PROGRAM T01_CONTROL
VAR
END_VAR

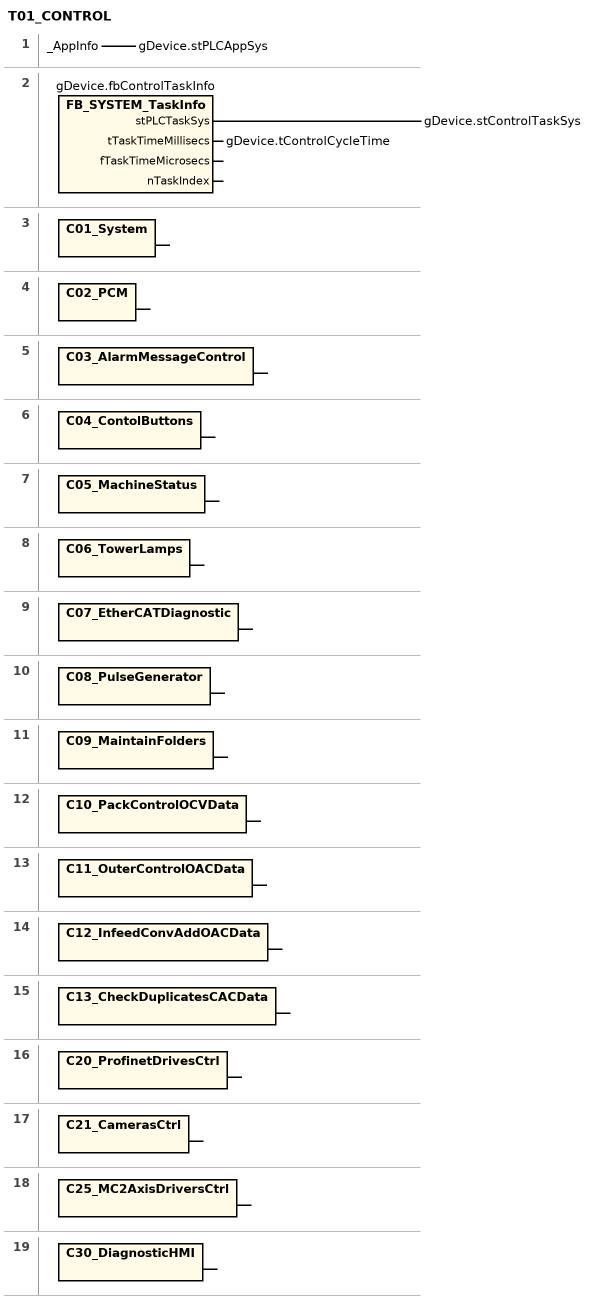
// NETWORK 1
gDevice.stPLCAppSys := _AppInfo;

// NETWORK 2
gDevice.fbControlTaskInfo(tTaskTimeMillisecs => gDevice.tControlCycleTime); // FB_SYSTEM_TaskInfo
gDevice.stControlTaskSys := gDevice.fbControlTaskInfo.stPLCTaskSys;

// NETWORK 3
C01_System();

// NETWORK 4
C02_PCM();

// NETWORK 5
C03_AlarmMessageControl();

// NETWORK 6
C04_ContolButtons();

// NETWORK 7
C05_MachineStatus();

// NETWORK 8
C06_TowerLamps();

// NETWORK 9
C07_EtherCATDiagnostic();

// NETWORK 10
C08_PulseGenerator();

// NETWORK 11
C09_MaintainFolders();

// NETWORK 12
C10_PackControlOCVData();

// NETWORK 13
C11_OuterControlOACData();

// NETWORK 14
C12_InfeedConvAddOACData();

// NETWORK 15
C13_CheckDuplicatesCACData();

// NETWORK 16
C20_ProfinetDrivesCtrl();

// NETWORK 17
C21_CamerasCtrl();

// NETWORK 18
C25_MC2AxisDriversCtrl();

// NETWORK 19
C30_DiagnosticHMI();

END_PROGRAM

(* stored: Version 1.1.0.1
   POU T01_CONTROL: Id {9c5412cc-d559-40cf-8c2c-a4222aa73aa8}, SpecialFunc None *)
